{attribute 'linkalways'} 
{attribute 'no_explicit_call' := 'This FB is a CLASS and must be accessed using methods or properties'}
{attribute 'enable_dynamic_creation'}
FUNCTION_BLOCK _TcVnVector2_LREAL EXTENDS AliasDatatypeBase
VAR
	localData : TcVnVector2_LREAL;
	activeData : REFERENCE TO TcVnVector2_LREAL REF= localData;
	aliasBaseDatatype : _Array0to1OfLREAL;
END_VAR

PROPERTY PUBLIC Address : PVOID
GET
Address := ADR(activeData);
END_GET
END_PROPERTY

METHOD PUBLIC ClearReference
VAR_INPUT
END_VAR
activeData REF= localData;
SetBaseDatatypeReference();
END_METHOD

METHOD PUBLIC Clone : I_Datatype
VAR
    pClone : POINTER TO _TcVnVector2_LREAL;
END_VAR
pClone := __NEW(_TcVnVector2_LREAL);
Clone := pClone^;
END_METHOD

METHOD FB_init : BOOL
VAR_INPUT
	bInitRetains : BOOL; // if TRUE, the retain variables are initialized (warm start / cold start)
	bInCopyCode : BOOL;  // if TRUE, the instance afterwards gets moved into the copy code (online change)
	//InitialValue : <type>; // if possible, not all values can be initialized
END_VAR
//localData := InitialValue; // if possible, not all values can be initialized
SetBaseDatatypeReference();
AddBaseDatatype(aliasBaseDatatype);
END_METHOD

PROPERTY PUBLIC Identifier : T_MAXSTRING
GET
Identifier := 'TcVnVector2_LREAL';
END_GET
END_PROPERTY

METHOD PUBLIC MakeReferenceTo
VAR_INPUT
	ReferenceTarget : REFERENCE TO TcVnVector2_LREAL;
END_VAR
activeData REF= ReferenceTarget;
SetBaseDatatypeReference();
END_METHOD

METHOD PROTECTED SetBaseDatatypeReference
VAR_INPUT
END_VAR
aliasBaseDatatype.MakeReferenceTo(activeData);
END_METHOD

PROPERTY PUBLIC Size : UDINT
GET
Size := SIZEOF(activeData);
END_GET
END_PROPERTY

METHOD TryMakeReferenceTo : BOOL
VAR_INPUT
	Target : I_Datatype;
END_VAR
VAR
	targetAsAlias : I_AliasDatatype;
	pTargetData : POINTER TO TcVnVector2_LREAL;
END_VAR
IF NOT Target.TryResolveAsAliasDatatype(targetAsAlias) THEN
	RETURN;
END_IF

IF targetAsAlias.Identifier <> Identifier THEN
	RETURN;
END_IF

pTargetData := Target.Address;
activeData REF= pTargetData^;
SetBaseDatatypeReference();
TryMakeReferenceTo := TRUE;
END_METHOD

PROPERTY PUBLIC Value : REFERENCE TO TcVnVector2_LREAL
GET
Value REF= activeData;
END_GET
END_PROPERTY

END_FUNCTION_BLOCK

(* stored: Version 1.1.0.1, ProductVersion 3.1.4024.13
   POU _TcVnVector2_LREAL: Id {7fdf00cb-7dc4-0b93-0daa-a31a822f7d35}, SpecialFunc None
   Folder Core: Id {673e1cd8-56df-0858-0f1e-30eff8117685}
   Folder Protected: Id {fa5c551f-8f66-0a05-2c46-36593a585b27}
   Folder Customize: Id {e0caee99-eace-0659-07b2-f32f68cca9a2}
   Folder Constructor: Id {87a0c14f-0b34-0815-3bf6-f27c88cd425a}
   Property Address: Id {e1135a65-3cf8-0fa3-174e-3b1875de3bd8}
   Get Get: Id {41d82723-ba7a-03b6-2462-c00bb374474e}
   Method ClearReference: Id {cdee6b84-afb5-09f1-0184-9641ba27bba6}
   Method Clone: Id {df9d0b6f-b5b9-00b6-3b43-8a667f7876aa}
   Method FB_init: Id {3594d155-fdea-085f-1dbb-749c45b01122}
   Property Identifier: Id {595bee1a-df36-001e-1adb-4e65851e7ca4}
   Get Get: Id {3e220020-70ed-087f-312d-4466d21c29e0}
   Method MakeReferenceTo: Id {dbc73afd-ac94-0921-2e57-39d52cae192e}
   Method SetBaseDatatypeReference: Id {76498ef8-ce29-0708-0ac2-3bf7c1af9201}
   Property Size: Id {1af54697-b319-00f8-0c3d-a047fc68786d}
   Get Get: Id {105f4945-a81c-0507-25ba-d16c8edc1f19}
   Method TryMakeReferenceTo: Id {e03afaeb-8dcf-0062-141a-c0792d587167}
   Property Value: Id {0eabe35b-41d7-0913-15fe-8c6a24ebc338}
   Get Get: Id {a4b8b692-4c96-08b2-38f1-0da383ed0f39} *)
